TYPE "FCP_CONTROL_WORD"
VERSION : 0.1
// Block: FCP_CONTROL_WORD
   STRUCT
      Reserved0 : Bool;
      Reserved1 : Bool;
      Reserved2 : Bool;
      Reserved3 : Bool;
      Reserved4 : Bool;
      Reserved5 : Bool;
      Reserved6 : Bool;
      Enable : Bool;
      Reserved8 : Bool;
      Reserved9 : Bool;
      Slave : Bool;
      ParGroup1 : Bool;
      Reserved12 : Bool;
      Reserved13 : Bool;
      Reserved14 : Bool;
      Reserved15 : Bool;
   END_STRUCT;

END_TYPE
